(* PLC project OOP_Curso, Beckhoff Automation GmbH TwinCAT PLC Control 3.5.13.21 *)
(* stored: creationDateTime 2023-09-23T11:43:14.2417075, modificationDateTime 2023-09-23T11:43:14.2511046 *)

INTERFACE I_Conexion
METHOD EstablecerConexion : BOOL
VAR_INPUT
END_VAR
END_METHOD
END_INTERFACE

FUNCTION_BLOCK ConexionEthernet IMPLEMENTS I_Conexion

VAR
//    rtMessageOutput: R_TRIG; (* Declaration *)
//    bFeedTooHigh: BOOL;
    udiAdsLogRes: UDINT;
END_VAR

            
          

METHOD EstablecerConexion : BOOL
                  //rtMessageOutput(CLK := bFeedTooHigh);
//IF rtMessageOutput.Q THEN 
    UdiAdsLogRes := ADSLOGDINT( msgCtrlMask := ADSLOG_MSGTYPE_HINT OR ADSLOG_MSGTYPE_MSGBOX, 
                    msgFmtStr := 'PLC Mensaje: estamos realizando una conexión por Ethernet: %d', dintArg:= 1);
//END_IF
                
END_METHOD
END_FUNCTION_BLOCK

FUNCTION_BLOCK ConexionSerial IMPLEMENTS I_Conexion

VAR
 //   rtMessageOutput: R_TRIG; (* Declaration *)
 //   bFeedTooHigh: BOOL;
    udiAdsLogRes: UDINT;
END_VAR

            
          

METHOD EstablecerConexion : BOOL
                  //rtMessageOutput(CLK := bFeedTooHigh);
//IF rtMessageOutput.Q THEN 
    UdiAdsLogRes := ADSLOGDINT( msgCtrlMask := ADSLOG_MSGTYPE_HINT OR ADSLOG_MSGTYPE_MSGBOX, 
                    msgFmtStr := 'PLC Mensaje: estamos realizando una conexión por Serial: %d', dintArg:= 1);
//END_IF
                
END_METHOD
END_FUNCTION_BLOCK

FUNCTION_BLOCK Dispositivo
VAR
	_conexion : I_Conexion;
END_VAR

            
          

METHOD establecerConexion 
VAR_INPUT
END_VAR
                  _conexion.EstablecerConexion();
                
END_METHOD

METHOD FB_init : BOOL
VAR_INPUT
	bInitRetains : BOOL; // if TRUE, the retain variables are initialized (warm start / cold start)
	bInCopyCode : BOOL;  // if TRUE, the instance afterwards gets moved into the copy code (online change)
	conexion : I_Conexion;
END_VAR
                  THIS^._conexion := conexion;
                
END_METHOD
END_FUNCTION_BLOCK

PROGRAM _28_SOLID_DIP
VAR
	Conexion_por_Serial : BOOL;
	Serial: ConexionSerial;
	Conexion_Serial : Dispositivo(conexion:= Serial);
	
	Conexion_por_Ethernet : BOOL;
	Ethernet : ConexionEthernet;
	Conexion_Ethernet : Dispositivo(conexion:= Ethernet);
END_VAR

            
IF Conexion_por_Serial THEN 
 Conexion_Serial.establecerConexion();
 Conexion_por_Serial:= FALSE;
END_IF

IF Conexion_por_Ethernet THEN 
 Conexion_Ethernet.establecerConexion();
 Conexion_por_Ethernet:= FALSE;
END_IF


          
END_PROGRAM
